// TIA Portal V17 export
// export: Created 2022-07-05T08:45:17.8555581Z, ExportSetting WithDefaults, DisplayName Totally Integrated Automation Portal, DisplayVersion V17, DisplayName TIA Portal Openness, DisplayVersion V17, DisplayName TIA Portal Version Control Interface, DisplayVersion V17, DisplayName STEP 7 Professional, DisplayVersion V17, DisplayName STEP 7 Safety, DisplayVersion V17, DisplayName WinCC Advanced, DisplayVersion V17
TYPE "OpcUaClientInterface.methodList.Method.Inputs"
// stored: IsFailsafeCompliant false
   STRUCT
      DateTime { ExternalAccessible := 'False'; ExternalVisible := 'False'; ExternalWritable := 'False'} : LDT;
   END_STRUCT;
END_TYPE
